# EPICS substitutions: exampleApp/Db/user.substitutions
# Example substitutions file

file "db/dbExample1.db" {
    { user = "mrippa" }
}

file db/dbExample2.db {
    pattern { user, no, scan }
        { "mrippa", 1, "1 second" }
        { "mrippa", 2, "2 second" }
        { "mrippa", 3, "5 second" }
}
